(* IEC 61131-3 sources: ae-motion-tiax/src/_internal, 3 files *)

(* ---- AxisCtrlTypes.st ---- *)
NAMESPACE Motion

    TYPE
        AxisData : STRUCT
            enabled : BOOL;
            homed : BOOL;
            cmd : AxisCmd;
        END_STRUCT;
    END_TYPE

    TYPE
        AxisCmd : INT (
            NONE := 0,
            ENABLE := 1,
            DISABLE := 2,
            STOP := 3,
            JOG := 4,
            POS_RELATIVE := 5,
            POS_ABSOLUTE := 6) := NONE;
    END_TYPE

END_NAMESPACE

(* ---- PosAxisCtrl.st ---- *)
USING Siemens.Simatic.S71500.MotionControl.Native;
NAMESPACE Motion

    CLASS PUBLIC PosAxisCtrl EXTENDS SpeedAxisCtrl

        VAR PROTECTED
            _mcHome         : MC_HOME;
            _mcMoveRel      : MC_MOVERELATIVE;
            _mcMoveAbs      : MC_MOVEABSOLUTE;
        END_VAR

        METHOD PUBLIC OVERRIDE SetAxis : BOOL
            VAR_INPUT
                axisDB : DB_ANY;
            END_VAR
            _axisDB := axisDB;
            SetAxis := THIS.RefToAxisIsValid();
        END_METHOD

        METHOD PUBLIC OVERRIDE ResetCmds
            SUPER.ResetCmds();
            _mcHome.Execute := FALSE;
            _mcMoveRel.Execute := FALSE;
            _mcMoveAbs.Execute := FALSE;
        END_METHOD

        METHOD PUBLIC HomeAxis
            VAR_INPUT
                position : LREAL;
                homingMode : INT;
            END_VAR
            _mcHome.Mode := homingMode;
            _mcHome.Position := position;
            _mcHome.Execute := TRUE;
        END_METHOD

        METHOD PUBLIC PosRelative
            VAR_INPUT
                distance : LREAL;
                velocity : LREAL;
                acceleration : LREAL;
                deceleration : LREAL;
                jerk : LREAL;
            END_VAR
            _mcMoveRel.Execute := TRUE;
            _mcMoveRel.Distance := distance;
            _mcMoveRel.velocity := velocity;
            _mcMoveRel.Acceleration := acceleration;
            _mcMoveRel.Deceleration := deceleration;
            _axisData.cmd := AxisCmd#POS_RELATIVE;
        END_METHOD

        METHOD PUBLIC PosAbsolute
            VAR_INPUT
                position : LREAL;
                velocity : LREAL;
                acceleration : LREAL;
                deceleration : LREAL;
                jerk : LREAL;
                direction : INT;
            END_VAR
            _mcMoveAbs.Execute := TRUE;
            _mcMoveAbs.Position := position;
            _mcMoveAbs.velocity := velocity;
            _mcMoveAbs.Acceleration := acceleration;
            _mcMoveAbs.Deceleration := deceleration;
            _mcMoveAbs.Jerk := jerk;
            IF direction > 0 THEN
                _mcMoveAbs.Direction := direction;
            ELSE
                _mcMoveAbs.Direction := 1;
            END_IF;
            _axisData.cmd := AxisCmd#POS_ABSOLUTE;
        END_METHOD

        METHOD PUBLIC OVERRIDE CyclicCall
            VAR_TEMP
                _axisAsPos      : REF_TO TO_PositioningAxis;
            END_VAR
            SUPER.CallMcBlocksSpeedAxis();
            THIS.CallMcBlocksPosAxis();
            _axisAsPos := AsPositioningAxisRef(_axisDB);
        END_METHOD

        METHOD PROTECTED CallMcBlocksPosAxis
            VAR_TEMP
                _axisAsPos      : REF_TO TO_PositioningAxis;
                _axisAsAxis     : REF_TO TO_Axis;
            END_VAR
            _axisAsPos := AsPositioningAxisRef(_axisDB);
            _axisAsAxis := _axisAsPos;
            IF _axisAsPos = NULL THEN
                RETURN;
            ELSE
                _mcHome(Axis := _axisAsAxis^);
                _mcMoveRel(Axis := _axisAsPos^);
                _mcMoveAbs(Axis := _axisAsPos^);

                IF _mcHome.Done THEN
                    _axisData.cmd := AxisCmd#NONE;
                    _mcHome.Execute := FALSE;
                END_IF;

                IF _mcMoveRel.Done OR _mcMoveRel.CommandAborted THEN
                    _mcMoveRel.Execute := FALSE;
                END_IF;

                IF _mcMoveAbs.Done OR _mcMoveAbs.CommandAborted THEN
                    _mcMoveAbs.Execute := FALSE;
                END_IF;
                _axisData.homed := _axisAsPos^.StatusWord.%X5;
            END_IF;
        END_METHOD

        METHOD PUBLIC OVERRIDE RefToAxisIsValid : BOOL
            VAR_TEMP
                _axisAsPos    : REF_TO TO_PositioningAxis;
            END_VAR
            _axisAsPos := AsPositioningAxisRef(_axisDB);
                RefToAxisIsValid := _axisAsPos <> NULL;
        END_METHOD

    END_CLASS

END_NAMESPACE

(* ---- SpeedAxisCtrl.st ---- *)
USING Siemens.Simatic.S71500.MotionControl.Native;
NAMESPACE Motion

    CLASS PUBLIC SpeedAxisCtrl

        VAR PROTECTED
            _mcPower    : MC_POWER;
            _mcJog      : MC_MOVEJOG;
            _mcHalt     : MC_HALT;
            _mcMoveVel  : MC_MOVEVELOCITY;
            _axisData   : AxisData;
            _axisDB : DB_ANY;
        END_VAR

        METHOD PUBLIC SetAxis : BOOL
            VAR_INPUT
                axisDB : DB_ANY;
            END_VAR
            _axisDB := axisDB;
            SetAxis := THIS.RefToAxisIsValid();
        END_METHOD

        METHOD PUBLIC ResetCmds
            _mcHalt.Execute := FALSE;
            _mcMoveVel.Execute := FALSE;
        END_METHOD

        METHOD PUBLIC EnableAxis
            VAR_INPUT
                startMode : INT;
            END_VAR
            _mcPower.StartMode := startMode;
            _mcPower.Enable := TRUE;
            _axisData.cmd := AxisCmd#ENABLE;
        END_METHOD

        METHOD PUBLIC DisableAxis
            VAR_INPUT
                stopMode : INT;
            END_VAR
            _mcPower.StopMode := stopMode;
            _mcPower.Enable := FALSE;
            _axisData.cmd := AxisCmd#DISABLE;
        END_METHOD

        METHOD PUBLIC StopAxis
            VAR_INPUT
                deceleration : LREAL;
                jerk : LREAL;
                abortAcceleration : BOOL;
            END_VAR
            _mcHalt.Deceleration := deceleration;
            _mcHalt.Jerk := jerk;
            _mcHalt.AbortAcceleration := abortAcceleration;
            _mcHalt.Execute := TRUE;
            _axisData.cmd := AxisCmd#STOP;
        END_METHOD

        METHOD PUBLIC MoveVelocity
            VAR_INPUT
                velocity : LREAL;
                acceleration : LREAL;
                deceleration : LREAL;
                jerk : LREAL;
                direction : INT;
                maintainCurrentVel : BOOL;
            END_VAR

            _mcMoveVel.velocity := velocity;
            _mcMoveVel.Acceleration := acceleration;
            _mcMoveVel.Deceleration := deceleration;
            _mcMoveVel.Jerk := jerk;
            _mcMoveVel.direction := direction;
            _mcMoveVel.Current := maintainCurrentVel;
            _mcMoveVel.Execute := TRUE;
        END_METHOD

        METHOD PUBLIC GetAxisStatus : AxisData
            GetAxisStatus := _axisData;
        END_METHOD

        METHOD PUBLIC CyclicCall
            THIS.CallMcBlocksSpeedAxis();
            _axisData.enabled := _mcPower.Status;
        END_METHOD

        METHOD PROTECTED CallMcBlocksSpeedAxis
            VAR_TEMP
                _axisAsSpeed    : REF_TO TO_SpeedAxis;
                _axisAsAxis     : REF_TO TO_Axis;
            END_VAR

            IF NOT THIS.RefToAxisIsValid() THEN
                RETURN;
            ELSE
                _axisAsSpeed := AsSpeedAxisRef(_axisDB);
                _axisAsAxis := AsAxisRef(_axisDB);
                _mcPower(Axis := _axisAsAxis^);
                _mcHalt(Axis := _axisAsSpeed^);
                _mcJog(Axis := _axisAsSpeed^);
                _mcMoveVel(Axis := _axisAsSpeed^);

                IF _mcHalt.Done THEN
                    _axisData.cmd := AxisCmd#NONE;
                    _mcHalt.Execute := FALSE;
                END_IF;

                IF _mcMoveVel.CommandAborted THEN
                    _axisData.cmd := AxisCmd#NONE;
                    _mcMoveVel.Execute := FALSE;
                END_IF;
            END_IF;
        END_METHOD

        METHOD PUBLIC RefToAxisIsValid : BOOL
            VAR_TEMP
                _axisAsSpeed    : REF_TO TO_SpeedAxis;
            END_VAR
                _axisAsSpeed := AsSpeedAxisRef(_axisDB);
                RefToAxisIsValid := _axisAsSpeed <> NULL;
        END_METHOD

    END_CLASS

END_NAMESPACE
